INTERFACE I_Enumerator EXTENDS __SYSTEM.IQueryInterface

// Gets an item in the collection at current positon of the enumerator.
METHOD Current : I_Enumerator
VAR_INPUT
	Item : ANY;
END_VAR
END_METHOD

// Gets an item in the collection at current positon of the enumerator as a string.
METHOD Current_As_String : I_Enumerable
VAR_INPUT
	sItem : REFERENCE TO STRING;
END_VAR
END_METHOD

// Releases resources allocated to the enumerator. Returns TRUE if successful.
METHOD Dispose : BOOL
VAR_INPUT
END_VAR
END_METHOD

// Advances the enumerator to the next item of the collection.
METHOD Next : BOOL
VAR_INPUT
END_VAR
END_METHOD

// Sets the enumerator to its initial position, which is before the first element in the collection.
METHOD Reset : I_Enumerator
END_METHOD

END_INTERFACE

(* stored: Version 1.1.0.1
   Itf I_Enumerator: Id {a65c5349-dfe5-0d69-378a-c0cbf28cab83}
   Method Current: Id {250f9020-9d82-0b8b-15e1-26e02378b56a}
   Method Current_As_String: Id {a8ff4bf3-e198-0177-1405-e9bdfab25837}
   Method Dispose: Id {dc20f7c7-7c9d-0e1f-0fa1-2b9cc45712f7}
   Method Next: Id {4e96be85-59b1-043e-1dcf-bc0ac23018f0}
   Method Reset: Id {01e8f251-faba-035a-0ecd-a225a9150b1f} *)
